PROGRAM MAIN
VAR
	Running				: BYTE;
	TimeAlive			: TON;
	TimeAliveSeconds	: INT;

END_VAR



// ======================================================================== //
//																			//
//					Beckhoff 2-Tile xPlanar Program							//
//																			//
//					Last Updated: 19-MAR-2025								//
//					Last Programmer: Ben Sturdy								//
//																			//
// ======================================================================== //


Running := Running + 1;


// Time the system has been in run mode (in seconds)
TimeAlive(IN := NOT TimeAlive.Q, PT := T#1S);
IF TimeAlive.Q THEN
	TimeAliveSeconds := TimeAliveSeconds + 1;
END_IF


xPlanarProgram();


CoeToPlc();

END_PROGRAM

(* stored: Version 1.1.0.1, ProductVersion 3.1.4024.12
   POU MAIN: Id {92246147-67ee-43d2-9056-44db244479e8}, SpecialFunc None *)
